// TwinCAT 3 PLC project Library01
// Title: MyLibrary01
// Company: MyCompany
// ProjectVersion: 2.0.0.0
// ProgramVersion: 3.1.4020.2
// libraries:
//   Tc2_Standard, * (Beckhoff Automation GmbH)
//   Tc2_System, * (Beckhoff Automation GmbH)
//   Tc3_Module, * (Beckhoff Automation GmbH)
// project tree:
//   DUTs/ E_Foo.TcDUT, ST_Foo.TcDUT
//   GVLs/ GVL01.TcGVL
//   / PlcTask.TcTTO (not stored)
//   POUs/ FB_Foo.TcPOU, I_Foo.TcIO
//   Version/ Global_Version.TcGVL
// real-time tasks:
//   TASK PlcTask: cycle T#10ms, priority 20, ADS port 350

// ---- DUTs/E_Foo.TcDUT
// {attribute 'qualified_only'}
// {attribute 'strict'}
TYPE E_Foo :
(
	eRed := 0,
	eBlue := 1,
	eGreen := 2
);
END_TYPE

// ---- DUTs/ST_Foo.TcDUT
TYPE ST_Foo :
STRUCT
	bVal01	:	BOOL;
	bVal02	:	BOOL;
END_STRUCT
END_TYPE

// ---- GVLs/GVL01.TcGVL
VAR_GLOBAL
	var01		:	INT;
END_VAR

// ---- Version/Global_Version.TcGVL
{attribute 'TcGenerated'}
// This function has been automatically generated from the project information.
VAR_GLOBAL CONSTANT
	{attribute 'const_non_replaced'}
	{attribute 'linkalways'}
	stLibVersion_MyLibrary01 : ST_LibVersion := (iMajor := 2, iMinor := 0, iBuild := 0, iRevision := 0, sVersion := '2.0.0.0');
END_VAR

// ---- POUs/I_Foo.TcIO
INTERFACE I_Foo

METHOD DoSomething : BOOL
VAR_INPUT
END_VAR
END_METHOD

END_INTERFACE

// ---- POUs/FB_Foo.TcPOU
FUNCTION_BLOCK PUBLIC FB_Foo
VAR_INPUT
END_VAR
VAR_OUTPUT
END_VAR
VAR
END_VAR

END_FUNCTION_BLOCK
